(* PLC project Unnamed, Unknown Unnamed 1 *)
(* stored: creationDateTime 2025-12-12T07:30:42, modificationDateTime 2025-12-16T19:31:49 *)

PROGRAM program0
  VAR
    BOTON_ARRANQUE AT %IX0.0 : BOOL;
    BOTON_PARADA AT %IX0.2 : BOOL;
    MOTOR_CINTA AT %QX1.0 : BOOL;
    VALVULA1_IN1 AT %QX0.2 : BOOL;
    VALVULA1_IN2 AT %QX0.3 : BOOL;
    VALVULA2_IN1 AT %QX0.0 : BOOL;
    VALVULA2_IN2 AT %QX0.1 : BOOL;
    VALVULA3_IN1 AT %QX0.5 : BOOL;
    VALVULA3_IN2 AT %QX0.6 : BOOL;
    SENSOR_IR_1 AT %IX2.7 : BOOL;
  END_VAR
  VAR
    TON0 : TON;
    TON1 : TON;
    TON2 : TON;
    TON4 : TON;
    TP0 : TP;
  END_VAR

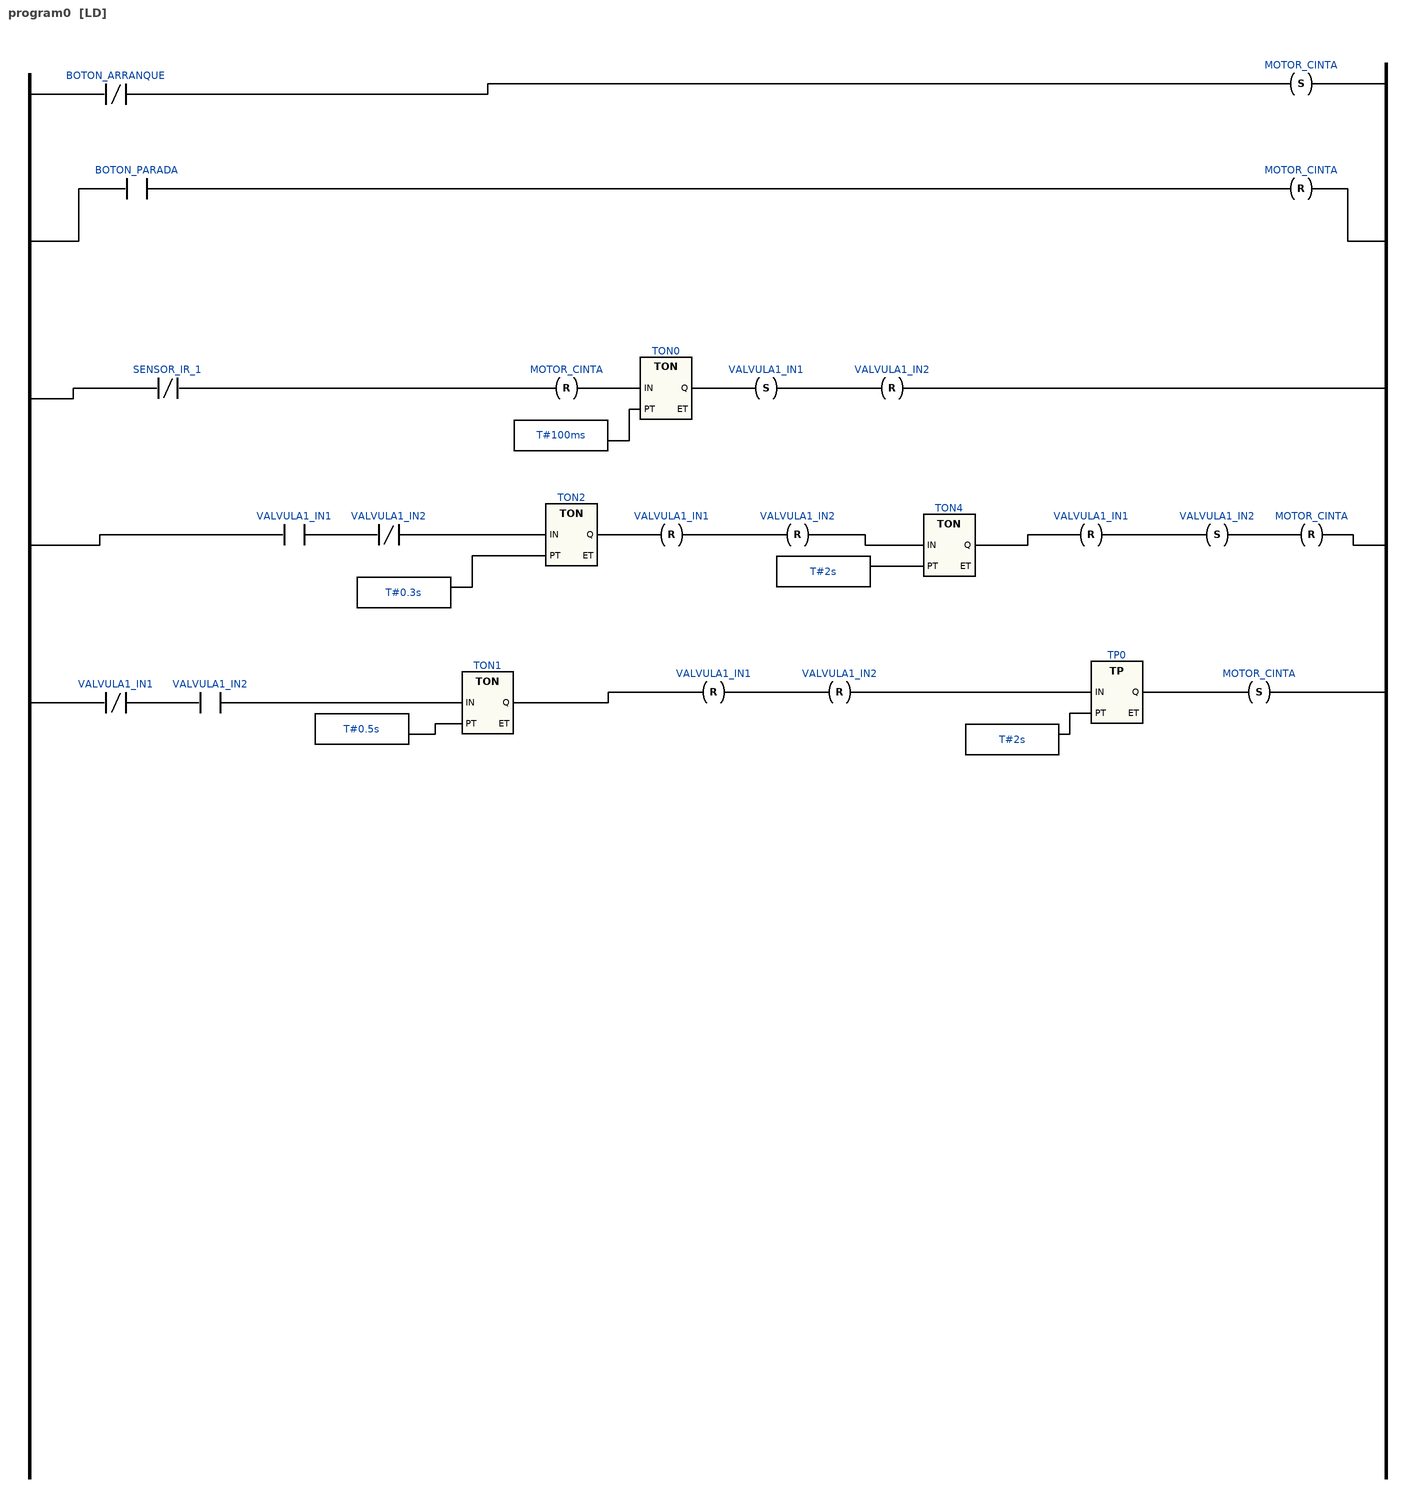
(* LD diagram, written out as Structured Text *)
IF NOT BOTON_ARRANQUE THEN MOTOR_CINTA := TRUE; END_IF;
IF BOTON_PARADA THEN MOTOR_CINTA := FALSE; END_IF;
IF NOT SENSOR_IR_1 THEN MOTOR_CINTA := FALSE; END_IF;
TON0(IN := NOT SENSOR_IR_1, PT := T#100ms);
IF TON0.Q THEN VALVULA1_IN1 := TRUE; END_IF;
IF TON0.Q THEN VALVULA1_IN2 := FALSE; END_IF;
TON2(IN := VALVULA1_IN1 AND NOT VALVULA1_IN2, PT := T#0.3s);
IF TON2.Q THEN VALVULA1_IN1 := FALSE; END_IF;
IF TON2.Q THEN VALVULA1_IN2 := FALSE; END_IF;
TON4(IN := TON2.Q, PT := T#2s);
IF TON4.Q THEN VALVULA1_IN2 := TRUE; END_IF;
IF TON4.Q THEN VALVULA1_IN1 := FALSE; END_IF;
TON1(IN := NOT VALVULA1_IN1 AND VALVULA1_IN2, PT := T#0.5s);
IF TON1.Q THEN VALVULA1_IN2 := FALSE; END_IF;
IF TON1.Q THEN VALVULA1_IN1 := FALSE; END_IF;
IF TON4.Q THEN MOTOR_CINTA := FALSE; END_IF;
TP0(IN := TON1.Q, PT := T#2s);
IF TP0.Q THEN MOTOR_CINTA := TRUE; END_IF;
END_PROGRAM

CONFIGURATION Config0
  RESOURCE Res0 ON PLC
    TASK task0(INTERVAL := T#20ms, PRIORITY := 0);
    PROGRAM instance0 WITH task0 : program0;
  END_RESOURCE
END_CONFIGURATION
